// TIA Portal project "HMI Demo" (V14)
// Práctica de demostrativa del uso de pantalla táctil y aplicación PC.

(* hardware
DEVICE "S7-1200 station_1"  S7-1200 Station
   slot 0: "Rack_0"  S7-1200 Rack  Rack  V1.0
   slot 1: "Controller"  CPU 1214C DC/DC/DC  6ES7 214-1AG40-0XB0  V4.2
DEVICE "Display_HMI"  TP700 Comfort
   slot 0: "TP700 Comfort"  TP700 Comfort  6AV2 124-0GC01-0AX0  14.0.1.0
   slot 1: "HMI_RT_1"  TP700 Comfort  6AV2 124-0GC01-0AX0  14.0.1.0
   slot 5: "Display_HMI.IE_CP_1"  PROFINET Interface  14.0.1.0
      slot 1: "PROFINET Interface_1"  PROFINET Interface
         slot 1: "Port_1"  Port
         slot 2: "Port_2"  Port
   slot 7: "Display_HMI.MPI/DP_CP_1"  MPI/DP Interface  14.0.1.0
*)

// ===== PLC "Controller"  CPU 1214C DC/DC/DC =====

VAR_GLOBAL   // PLC tag table "Default tag table"
   "sensor" AT %IW64 : Int;
   "variable_tmp" AT %MD4 : Real;
   "Current Temperature" AT %MW8 : Int;
   "Max Temperature" AT %IW10 : Int;
   "Min Temperature" AT %IW12 : Int;
   "Warning Text" AT %MW14 : Int;
   "Warning" AT %Q0.0 : Bool;
   "temp0" AT %M2.0 : Bool;
   "temp1" AT %M2.1 : Bool;
   "temp2" AT %M2.2 : Bool;
END_VAR

FUNCTION "Temperature Warnings" : Void   // FC1, LAD
{ S7_Optimized_Access := 'TRUE' }
VERSION : 0.1
   VAR_OUTPUT
      Warning : Bool;
      "Warning Text" : Int;
   END_VAR
   VAR_IN_OUT
      "Current Temperature" : Int;
      "Max Temperature" : Int;
      "Min Temperature" : Int;
   END_VAR
   VAR CONSTANT
      Tag1 : WString := WSTRING#'Heatstroke Warning';
      Tag2 : WString := WSTRING#'No Warning';
      Tag3 : WString := WSTRING#'Freeze Warning';
   END_VAR
   VAR_TEMP   // added for the SCL form of the ladder/FBD networks
      _w1 : Bool;
   END_VAR
BEGIN

REGION Network 1: Heatstroke Warning
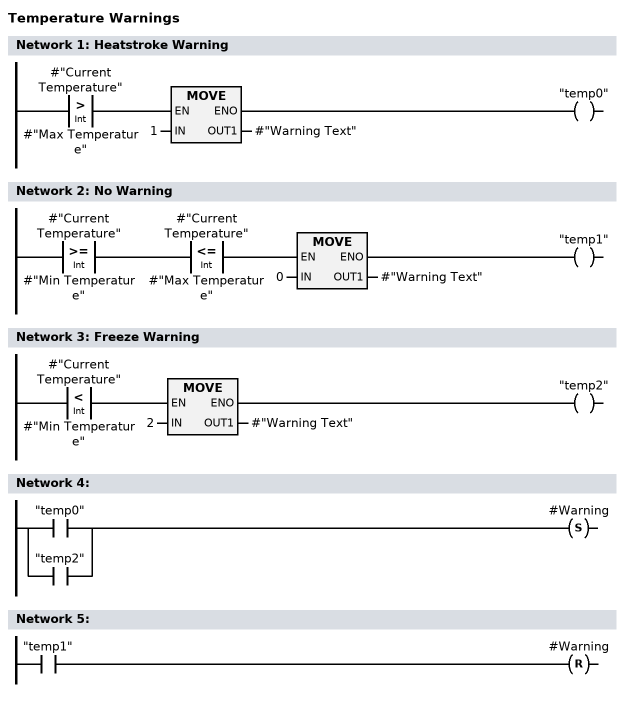
   RUNG wire#powerrail
      { S7_Templates := "SrcType := Int" } GT_Contact(in1 := #"Current Temperature", in2 := #"Max Temperature")
      Move(in := 1, out1 => #"Warning Text")
      Coil( "temp0" )
   END_RUNG
   // the same network as SCL:
   #_w1 := #"Current Temperature" > #"Max Temperature";
   IF #_w1 THEN #"Warning Text" := 1; END_IF;
   "temp0" := #_w1;
END_REGION

REGION Network 2: No Warning
   RUNG wire#powerrail
      { S7_Templates := "SrcType := Int" } GE_Contact(in1 := #"Current Temperature", in2 := #"Min Temperature")
      { S7_Templates := "SrcType := Int" } LE_Contact(in1 := #"Current Temperature", in2 := #"Max Temperature")
      Move(in := 0, out1 => #"Warning Text")
      Coil( "temp1" )
   END_RUNG
   // the same network as SCL:
   #_w1 := (#"Current Temperature" >= #"Min Temperature") AND (#"Current Temperature" <= #"Max Temperature");
   IF #_w1 THEN #"Warning Text" := 0; END_IF;
   "temp1" := #_w1;
END_REGION

REGION Network 3: Freeze Warning
   RUNG wire#powerrail
      { S7_Templates := "SrcType := Int" } LT_Contact(in1 := #"Current Temperature", in2 := #"Min Temperature")
      Move(in := 2, out1 => #"Warning Text")
      Coil( "temp2" )
   END_RUNG
   // the same network as SCL:
   #_w1 := #"Current Temperature" < #"Min Temperature";
   IF #_w1 THEN #"Warning Text" := 2; END_IF;
   "temp2" := #_w1;
END_REGION

REGION Network 4
   RUNG wire#powerrail
      Contact( "temp0" )
      wire#w1
      S_Coil( #Warning )
   END_RUNG
   RUNG wire#powerrail
      Contact( "temp2" )
   END_RUNG wire#w1
   // the same network as SCL:
   IF "temp0" OR "temp2" THEN #Warning := TRUE; END_IF;
END_REGION

REGION Network 5
   RUNG wire#powerrail
      Contact( "temp1" )
      R_Coil( #Warning )
   END_RUNG
   // the same network as SCL:
   IF "temp1" THEN #Warning := FALSE; END_IF;
END_REGION
END_FUNCTION

FUNCTION "Temperature ADQ" : Void   // FC2, LAD
{ S7_Optimized_Access := 'TRUE' }
VERSION : 0.1
   VAR_INPUT
      "Temperature Sensor" : Int;
   END_VAR
   VAR_OUTPUT
      Temperature : Int;
   END_VAR
BEGIN

REGION Network 1
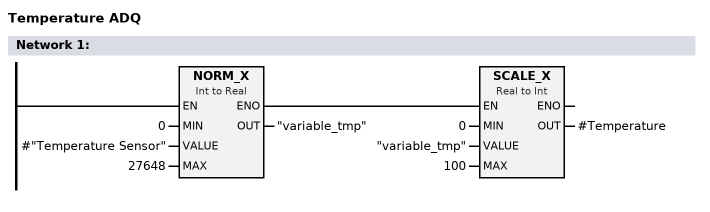
   RUNG wire#powerrail
      { S7_Templates := "[SrcType := Int, DestType := Real]" } Normalize(min := 0, value := #"Temperature Sensor", max := 27648, out => "variable_tmp")
      { S7_Templates := "[SrcType := Real, DestType := Int]" } Scale(min := 0, value := "variable_tmp", max := 100, out => #Temperature)
   END_RUNG
   // the same network as SCL:
   "variable_tmp" := NORM_X(MIN := 0, VALUE := #"Temperature Sensor", MAX := 27648);
   #Temperature := SCALE_X(MIN := 0, VALUE := "variable_tmp", MAX := 100);
END_REGION
END_FUNCTION

ORGANIZATION_BLOCK "Main"   // OB1, LAD, ProgramCycle
TITLE = "Main Program Sweep (Cycle)"
{ S7_Optimized_Access := 'TRUE' }
VERSION : 0.1
   VAR_INPUT
      Initial_Call : Bool;   // Initial call of this OB
      Remanence : Bool;   // =True, if remanent data are available
   END_VAR
BEGIN

REGION Network 1: Temperature Adquisition
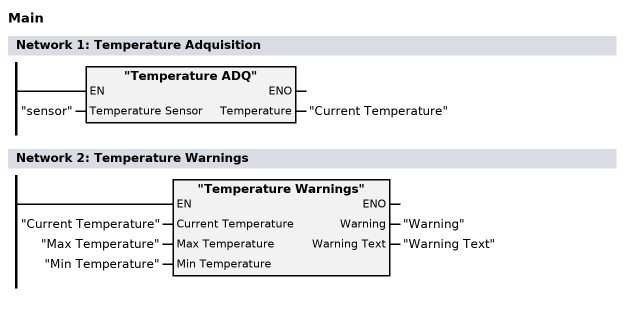
   RUNG wire#powerrail
      "Temperature ADQ"("Temperature Sensor" := "sensor", Temperature => "Current Temperature")
   END_RUNG
   // the same network as SCL:
   "Temperature ADQ"("Temperature Sensor" := "sensor", Temperature => "Current Temperature");
END_REGION

REGION Network 2: Temperature Warnings
   RUNG wire#powerrail
      "Temperature Warnings"("Current Temperature" := "Current Temperature", "Max Temperature" := "Max Temperature", "Min Temperature" := "Min Temperature", Warning => "Warning", "Warning Text" => "Warning Text")
   END_RUNG
   // the same network as SCL:
   "Temperature Warnings"("Current Temperature" := "Current Temperature",
                          "Max Temperature" := "Max Temperature",
                          "Min Temperature" := "Min Temperature",
                          Warning => "Warning",
                          "Warning Text" => "Warning Text");
END_REGION
END_ORGANIZATION_BLOCK

(* ===== HMI "HMI_RT_1" =====
system functions are stored by id; their names below are inferred from use
connection "HMI_Connection_1": ETHERNET, S7_1200_OMS

HMI tags "Default tag table"
   "Tag_ScreenNumber" : UInt, internal
   "Current Temperature HMI" : Int = PLC "Current Temperature" AT %MW8, 1 s
   "Max Temperature HMI" : Int = PLC "Max Temperature" AT %IW10, 1 s
   "Min Temperature HMI" : Int = PLC "Min Temperature" AT %IW12, 1 s
   "Warning_HMI" : Bool = PLC Warning AT %Q0.0, 1 s
   "Warning Text HMI" : Int = PLC "Warning Text" AT %MW14, 1 s

text list "Text_list_1": 1 'Heatstroke Warning'; 2..3 'No Warning'; 2 'Freeze Warning'

screen "Root screen" 800x420, template "Template_1"
   on GenerateScreen: SetTag("Tag_ScreenNumber", 1)
   TextField "HmiScreenItemData" at 0,319 size 429x25; Text 'Welcome to Display_HMI (TP700 Comfort)!'
   IOField "I/O field_1" at 376,150 size 96x32; FormatPattern s99999
      ProcessValue <- "Current Temperature HMI"
   TextField "Text field_1" at 376,114 size 198x23; Text 'Current Temperature'
   GraphicIOField "PlotLight_Round_R" at 613,92 size 50x50; PictureOn "PilotLight_Round_R_On_256c"; PictureOff "PilotLight_Round_R_Off_256c"
      ProcessValue <- "Warning_HMI"
   TextField "Text field_4" at 613,66 size 90x23; Text 'Warning?'
   TextField "Text field_5" at 613,155 size 128x23; Text 'Warning Text'
   Slider "Slider_1" at 66,59 size 80x230; Caption 'Max'
      ProcessValue <- "Max Temperature HMI"
   Slider "Slider_2" at 208,59 size 80x230; Caption 'Min'
      ProcessValue <- "Min Temperature HMI"
   Button "Button_1" at 567,194 size 183x32; TextOff 'No Warning'; TextOn 'Alarm!!'; TextList "Text_list_1"
      ProcessValue <- "Warning Text HMI"

Template "Template_1" 800x420
   Button "Exit" at 720,360 size 78x58; TextOff 'Exit'; PictureOff "ExitRuntime_TP700_Comfort_TR"; PictureOn "ExitRuntime_TP700_Comfort_TR"
      on Release: StopRuntime(0)
   Button "Template_Button" at 640,360 size 78x58; TextOff 'Text'
   Button "Template_Button_1" at 560,360 size 78x58; TextOff 'Text'
   Button "Template_Button_2" at 480,360 size 78x58; TextOff 'Text'
   Button "Template_Button_3" at 400,360 size 78x58; TextOff 'Text'
   Button "Template_Button_4" at 321,360 size 78x58; TextOff 'Text'
   Button "Template_Button_5" at 241,360 size 78x58; TextOff 'Text'
   Button "Template_Button_6" at 161,360 size 78x58; TextOff 'Text'
   Button "Alarms" at 81,360 size 78x58; TextOff 'Alarms'; PictureOff "AlarmDisplay_TP700_Comfort_TR"; PictureOn "AlarmDisplay_TP700_Comfort_TR"
      on Release: function_ef3f5d25("Alarm window_Unacknowledged", -1)
   Button "Start screen" at 1,360 size 78x58; TextOff 'Start screen'; PictureOff "NavigateHome_TP700_Comfort_TR"; PictureOn "NavigateHome_TP700_Comfort_TR"
      on Release: ActivateScreen("Root screen", 0)
*)